FUNCTION_BLOCK FB_BMS
VAR_OUTPUT
	PowerStatus: eHVDC_Powerstatus := 0;
END_VAR
VAR_INPUT
	Set : st_BMS_Set;
END_VAR

VAR_OUTPUT
	BMSGet: st_BMS_GetStatus;
END_VAR

VAR	
	FBState				:	ePOUState;
	IO					:	FB_BMS_IO;
	HWControl			:	st_BMS_IO;
	
	InitTimeout			: 	TON := (PT:=T#3S);
	
	BMS_230V_StartupTimer : TON := (PT := TIME#3S0MS);
	BMS_24V_StartupTimer : TON := (PT := TIME#2S0MS);
	
	TempVar				: WORD;
	SFCInit				: BOOL := FALSE;
	SFCReset			: BOOL := FALSE;
	
//	by_CommErrorCounter	:	BYTE	:=	0;
	b_MBComErrorActive	: 	BOOL 	:= FALSE;
	
	ResetBMS	:	Bool; 
	b_BMSShutdownRequested: BOOL;
	
	BMSReadIntervalTimer	 : TON := (PT := TIME#1S0MS);
END_VAR

(*
FB_BMS

Inputs
	Set.b_EnableBMS				:	BOOL;
		Start BMS SFC sequence and initializes BMS. False means full BMS powerdown, so no status logging.
		With HVDC enabled, setting this value to False has no effect. Only after HVDC powerdown this value is tested.
		
	Set.b_ClearFault				:	BOOL;
		Clear errors and warning in BMS system. Set to true to initiate reset. Value resets automatically to false.
	
	Set.b_HVDC_Required			: 	BOOL;
		Set by FB_internalPowersupply. True initiates and keeps HVDC on, False initiates and retains powerdown

Outputs
	BMSGET
		-Some general status info
		-BATTinfo	struct with main operation battery data
		-MBMU_Status 	struct with detailed MBMU data
		-SBMU			Struct with detailed data per SBMU
		-Events			Warnings & Errors as per Sunspec list.
*)

IO(HWControl:=HWControl);

BMSReadIntervalTimer(in:= not BMSReadIntervalTimer.Q);

//Reset ErrorActive before entering SFC. 
//any remaining error in the Modbus methods will set Erroractive again. 
//This is pushed to events in BMS_Diagnostics

//TEMPBMSHB();
//hv required not allowed if BMS not enabled
set.b_HVDC_Required := set.b_HVDC_Required AND Set.b_EnableBMS;
//shutdown allowed if hvdc is offline
b_BMSShutdownRequested := (NOT Set.b_EnableBMS) AND BMSGet.BattInfo.ui_BMS_PowerOnStatus <> ePowerOnStatus.On; 

//b_MBComErrorActive := FALSE;

IF FBState = ePOUState.EMSTOP THEN
	Set.b_HVDC_Required := FALSE;
END_IF

BMSSFC();


IF ResetBMS THEN
	Reset();
END_IF


BMS_Diagnostics();

ACTION aBMSPoweroff:
HWControl.b_BMS_230V_Enable := FALSE;
HWControl.b_BMS_24V_Enable := FALSE;

BMSGet.BattInfo.b_BMSHeartBeatOK := FALSE;
BMSGet.BattInfo.ui_BMS_PowerOnStatus := ePowerOnStatus.Off;
BMSGet.BattInfo.ui_BMS_Status := eBMS_Status.Off;

BMSGet.MBMU_Status.BatteryStatus.b_BMSHeartBeatOK := FALSE;
BMSGet.MBMU_Status.BatteryStatus.ui_BMS_PowerOnStatus := ePowerOnStatus.Off;
BMSGet.MBMU_Status.BatteryStatus.ui_BMS_Status := eBMS_Status.Off;

FBState := ePOUState.OFF;
END_ACTION

ACTION aBMSPowerOn:

//230V inverter requires some startup time. Start this first to init SBMU before MBMU
//This may not be needed, but the idea is to make sure the MBMU can reach the SBMU's at boot.
FBState := ePOUState.PowerUp;
HWControl.b_BMS_230V_Enable := TRUE;
BMS_230V_StartupTimer(IN:=HWControl.b_BMS_230V_Enable);

HWControl.b_BMS_24V_Enable := BMS_230V_StartupTimer.Q;
BMS_24V_StartupTimer(IN:=HWControl.b_BMS_24V_Enable);
END_ACTION

ACTION aClearFaults:
SFCTip := ClearBMSFaults();
END_ACTION

ACTION aDisableInsulationMonitor:
SFCTip := OpenInsulationSwitch(TRUE);
END_ACTION

ACTION aGetMBMUData:
SFCTip := GetMBMUData();
END_ACTION

ACTION aGetSBMUData:
SFCTip := GetSBMUData();
END_ACTION

ACTION aGetStaticData:

IF (TempVar=0) THEN
	IF GetMBMUStaticSystemData() THEN
		TempVar:=1;
	END_IF;
ELSE
	IF GetSBMUStaticSystemData(TempVar) THEN
		TempVar := TempVar+1;
	END_IF
	
	IF TempVar > 4 then//BMSGet.MBMU_Status.by_NumberOfSubSystems THEN
		TempVar:=0;
		SFCTip := TRUE;
	END_IF
END_IF
END_ACTION

ACTION aGetStatus:
IF GetSystemStatus() THEN
	IF FBState = ePOUState.PowerUp THEN FBState := ePOUState.Init; END_IF
	SFCTip := TRUE;
END_IF
END_ACTION

ACTION aInit:
TempVar := 0;
SFCReset := false;
END_ACTION

ACTION aSetDateTime:
SFCTip := SetBMSDateTime();
END_ACTION

ACTION aSetPowerMode:
SFCTip := SetPowerMode();
END_ACTION

ACTION aWatchdog:
IF FBState = ePOUState.Init THEN FBState := ePOUState.Normal; END_IF

SFCTip := BMSHeartBeat();
TempVar := 0;
END_ACTION

METHOD BMS_Diagnostics : BOOL
VAR
	
END_VAR

BMSGet.Events.b_COMMUNICATION_ERROR				:=	BMSGet.MBMU_Status.GeneralSBMUStatus[6].5 	//SBMU CCAN comm lost
												OR BMSGet.MBMU_Status.GeneralSBMUStatus[6].6 	//SBMU SCAN comm lost
												OR BMSGet.MBMU_Status.GeneralSBMUStatus[6].7	//SBMU MCAN comm lost
												OR BMSGet.MBMU_Status.MBMUStatus[0].6			//MBMU MCAN comm warning
												OR BMSGet.MBMU_Status.MBMUStatus[0].7			//MBMU MCAN comm Lost
												OR BMSGet.MBMU_Status.MBMUStatus[0].8			//SBMU EMS COMM lost
												OR BMSGet.MBMU_Status.MBMUStatus[3].4			//SBMU MBMU comm fault
												OR b_MBComErrorActive;					//One or more Modbus communication errors 
									
BMSGet.Events.b_OVER_TEMP_ALARM					:= BMSGet.MBMU_Status.GeneralSBMUStatus[2].1;	//single cell Overtemperature warning 4

BMSGet.Events.b_OVER_TEMP_WARNING				:= BMSGet.MBMU_Status.GeneralSBMUStatus[1].14	//single cell Overtemperature warning 1
												OR BMSGet.MBMU_Status.GeneralSBMUStatus[2].0; 	//single cell Overtemperature warning 2

BMSGet.Events.b_UNDER_TEMP_ALARM				:= FALSE; //no data

BMSGet.Events.b_UNDER_TEMP_WARNING				:= BMSGet.MBMU_Status.GeneralSBMUStatus[2].2	//single cell Undertemperature warning 1
												OR BMSGet.MBMU_Status.GeneralSBMUStatus[2].3 	//single cell Undertemperature warning 2
												OR BMSGet.MBMU_Status.GeneralSBMUStatus[2].4; 	//single cell Undertemperature warning 3

BMSGet.Events.b_OVER_CHARGE_CURRENT_ALARM		:= BMSGet.MBMU_Status.GeneralSBMUStatus[1].9;	//Charge Overcurrent warning 4

BMSGet.Events.b_OVER_CHARGE_CURRENT_WARNING		:= BMSGet.MBMU_Status.GeneralSBMUStatus[1].6	//Charge Overcurrent warning 1
												OR BMSGet.MBMU_Status.GeneralSBMUStatus[1].7 	//Charge Overcurrent warning 2
												OR BMSGet.MBMU_Status.GeneralSBMUStatus[1].8; 	//Charge Overcurrent warning 3
											
BMSGet.Events.b_OVER_DISCHARGE_CURRENT_ALARM	:= BMSGet.MBMU_Status.GeneralSBMUStatus[1].5;	//Discharge Overcurrent warning 4

BMSGet.Events.b_OVER_DISCHARGE_CURRENT_WARNING	:= BMSGet.MBMU_Status.GeneralSBMUStatus[1].2	//Discharge Overcurrent warning 1
												OR BMSGet.MBMU_Status.GeneralSBMUStatus[1].3 	//Discharge Overcurrent warning 2
												OR BMSGet.MBMU_Status.GeneralSBMUStatus[1].4; 	//Discharge Overcurrent warning 3
											
BMSGet.Events.b_OVER_VOLT_ALARM					:= BMSGet.MBMU_Status.GeneralSBMUStatus[0].6;	//Single cell extreme overVoltage warning

BMSGet.Events.b_OVER_VOLT_WARNING				:= BMSGet.MBMU_Status.GeneralSBMUStatus[0].0	//Single cell overVoltage warning 1
												OR BMSGet.MBMU_Status.GeneralSBMUStatus[0].1 	//Single cell overVoltage warning 2
												OR BMSGet.MBMU_Status.GeneralSBMUStatus[0].2 	//Single cell overVoltage warning 3
												OR BMSGet.MBMU_Status.GeneralSBMUStatus[0].8 	//Single rack overVoltage warning 1
												OR BMSGet.MBMU_Status.GeneralSBMUStatus[0].9; 	//Single rack overVoltage warning 2
												
BMSGet.Events.b_UNDER_VOLT_ALARM				:= BMSGet.MBMU_Status.GeneralSBMUStatus[0].7;	//Single cell extreme underVoltage warning

BMSGet.Events.b_UNDER_VOLT_WARNING				:= BMSGet.MBMU_Status.GeneralSBMUStatus[0].3	//Single cell underVoltage warning 1
												OR BMSGet.MBMU_Status.GeneralSBMUStatus[0].4 	//Single cell underVoltage warning 2
												OR BMSGet.MBMU_Status.GeneralSBMUStatus[0].5 	//Single cell underVoltage warning 3
												OR BMSGet.MBMU_Status.GeneralSBMUStatus[0].10 	//Single rack underVoltage warning 1
												OR BMSGet.MBMU_Status.GeneralSBMUStatus[0].11; //Single rack underVoltage warning 2
												
BMSGet.Events.b_UNDER_SOC_MIN_ALARM				:= BMSGet.MBMU_Status.GeneralSBMUStatus[6].14;	//r_SOC low warning 2

BMSGet.Events.b_UNDER_SOC_MIN_WARNING			:= BMSGet.MBMU_Status.GeneralSBMUStatus[6].13;	//r_SOC low warning 1

BMSGet.Events.b_OVER_SOC_MAX_ALARM				:= FALSE; //no data

BMSGet.Events.b_OVER_SOC_MAX_WARNING			:= FALSE; //no data

BMSGet.Events.b_VOLTAGE_IMBALANCE_WARNING		:= BMSGet.MBMU_Status.GeneralSBMUStatus[0].12;	//large voltage difference warning

BMSGet.Events.b_TEMPERATURE_IMBALANCE_ALARM		:= FALSE; //no data
												
BMSGet.Events.b_TEMPERATURE_IMBALANCE_WARNING	:= BMSGet.MBMU_Status.GeneralSBMUStatus[2].5	//Large temperature difference warning 1
												OR BMSGet.MBMU_Status.GeneralSBMUStatus[2].6 	//Large temperature difference warning 2
												OR BMSGet.MBMU_Status.GeneralSBMUStatus[2].7; 	//Large temperature difference warning 3
												
BMSGet.Events.b_CONTACTOR_ERROR					:= BMSGet.MBMU_Status.GeneralSBMUStatus[5].1	//Main positive relay sticking
												OR BMSGet.MBMU_Status.GeneralSBMUStatus[5].2 	//Main negative relay sticking
												OR BMSGet.MBMU_Status.GeneralSBMUStatus[5].3 	//Both main relays sticking
												OR BMSGet.MBMU_Status.GeneralSBMUStatus[5].4 	//Main positive relay open
												OR BMSGet.MBMU_Status.GeneralSBMUStatus[5].5 	//Main negative relay open
												OR BMSGet.MBMU_Status.GeneralSBMUStatus[6].15; //HV open circuit warning
												
BMSGet.Events.b_FAN_ERROR						:= BMSGet.MBMU_Status.GeneralSBMUStatus[5].7;	//main control box fan warning

BMSGet.Events.b_GROUND_FAULT					:= FALSE; //no data

BMSGet.Events.b_OPEN_DOOR_ERROR					:= FALSE; //no data

BMSGet.Events.b_CURRENT_IMBALANCE_WARNING		:= FALSE; //no data

BMSGet.Events.b_OTHER_ALARM						:= BMSGet.MBMU_Status.GeneralSBMUStatus[0].13	//Invalid voltage warning
												OR BMSGet.MBMU_Status.GeneralSBMUStatus[1].10 	//Current sensor fault
												OR BMSGet.MBMU_Status.GeneralSBMUStatus[2].15 //single temperature sampling abnormal value warning
												OR BMSGet.MBMU_Status.GeneralSBMUStatus[3].0 	//multiple temperature sampling abnormal value warning
												OR BMSGet.MBMU_Status.GeneralSBMUStatus[4].9 	//CSC supply abnormal
												OR BMSGet.MBMU_Status.GeneralSBMUStatus[4].10 	//SBMU supply abnormal
												OR BMSGet.MBMU_Status.GeneralSBMUStatus[4].14 	//MSD warning
												OR BMSGet.MBMU_Status.GeneralSBMUStatus[4].15 	//rack fuse warning
												OR BMSGet.MBMU_Status.GeneralSBMUStatus[6].11 	//cell balance circuit short
												OR BMSGet.MBMU_Status.GeneralSBMUStatus[7].3 	//precharching failed twice
												OR BMSGet.MBMU_Status.MBMUStatus[1].7 			//estop fault
												OR BMSGet.MBMU_Status.MBMUStatus[3].3; 		//MBMU 24V fault
												
BMSGet.Events.b_OTHER_WARNING					:= BMSGet.MBMU_Status.MBMUStatus[0].0 			//insulation warning
												OR BMSGet.MBMU_Status.MBMUStatus[1].10 		//rack fan warning
												OR BMSGet.MBMU_Status.MBMUStatus[3].7;			//TMS warning
												
BMSGet.Events.b_CONFIGURATION_ALARM				:= BMSGet.MBMU_Status.GeneralSBMUStatus[5].0	//rack isolate switch warning
												OR BMSGet.MBMU_Status.GeneralSBMUStatus[5].6 	//battery rack door fault
												OR BMSGet.MBMU_Status.GeneralSBMUStatus[5].9 	//rack fire system level 1 fault
												OR BMSGet.MBMU_Status.GeneralSBMUStatus[5].10 	//smoke detector contact open
												OR BMSGet.MBMU_Status.GeneralSBMUStatus[5].11 	//temp detector contact open
												OR BMSGet.MBMU_Status.GeneralSBMUStatus[5].14 	//aerosol warning
												OR BMSGet.MBMU_Status.GeneralSBMUStatus[6].0 	//rack fire system level 2 fault
												OR BMSGet.MBMU_Status.GeneralSBMUStatus[6].10 	//SBMU TMS CCAN comm lost with hv on
												OR BMSGet.MBMU_Status.GeneralSBMUStatus[7].0 	//lvl 3 fault tms
												OR BMSGet.MBMU_Status.GeneralSBMUStatus[7].1 	//TMS mode conflict
												OR BMSGet.MBMU_Status.GeneralSBMUStatus[7].2 	//TMS warning
												OR BMSGet.MBMU_Status.GeneralSBMUStatus[8].0 	//Thermal runaway caused fire
												OR BMSGet.MBMU_Status.MBMUStatus[0].1	 		//Insulation fault
												OR BMSGet.MBMU_Status.MBMUStatus[0].2			//Insulation error
												OR BMSGet.MBMU_Status.MBMUStatus[0].3 			//Less HV racks than expected
												OR BMSGet.MBMU_Status.MBMUStatus[0].9			//IMM comm fault
												OR BMSGet.MBMU_Status.MBMUStatus[0].10 		//Air conditioning comm fault
												OR BMSGet.MBMU_Status.MBMUStatus[0].11			//TMS comm fault
												OR BMSGet.MBMU_Status.MBMUStatus[0].13			//TMS comm fault lvl 2
												OR BMSGet.MBMU_Status.MBMUStatus[0].14 		//TMS mode conflict
												OR BMSGet.MBMU_Status.MBMUStatus[0].15			//TMS comm fault level 1
												OR BMSGet.MBMU_Status.MBMUStatus[1].3	 		//AUX power DCDC failure
												OR BMSGet.MBMU_Status.MBMUStatus[1].4			//Fire system fault lvl 1
												OR BMSGet.MBMU_Status.MBMUStatus[1].5 			//Fire system fault lvl 2
												OR BMSGet.MBMU_Status.MBMUStatus[1].6			//Fire system failure warning
												OR BMSGet.MBMU_Status.MBMUStatus[1].8	 		//client estop fault
												OR BMSGet.MBMU_Status.MBMUStatus[1].9			//rack door fault
												OR BMSGet.MBMU_Status.MBMUStatus[1].12;		//smoke ex fan body fault
								
BMSGet.Events.b_CONFIGURATION_WARNING			:= BMSGet.MBMU_Status.GeneralSBMUStatus[6].8	//SBMU TMS CCAN comm lost
												OR BMSGet.MBMU_Status.MBMUStatus[0].12	 		//TMS comm warning
												OR BMSGet.MBMU_Status.MBMUStatus[1].0			//SPD failure
												OR BMSGet.MBMU_Status.MBMUStatus[1].1 			//Aux power DCDC failure
												OR BMSGet.MBMU_Status.MBMUStatus[1].2			//AUX power DCDC failure
												OR BMSGet.MBMU_Status.MBMUStatus[1].6 			//Fire system failure warning
												OR BMSGet.MBMU_Status.MBMUStatus[1].11;		//Smoke exhaust fan body warning
END_METHOD

METHOD BMSHeartBeat : BOOL

VAR_INST
	WriteReg		:	FB_MBWriteSingleReg;
	ReadReg			:	FB_MBReadRegs;
	
	readbCommBusy		:	BOOL;
	readbComError		:	BOOL;
	readerrID			:	UDINT;
	
	WritebCommBusy		:	BOOL;
	WritebComError		:	BOOL;
	WriteerrID			:	UDINT;
	
	ReadDone			:	F_Trig;
	ReadOK				: 	BOOL;
	WriteDone			:	F_Trig;
	WriteOK				: 	BOOL;
	
	ComTimer		:	Ton := (PT := TIME#0S200MS);
	
	OldValue		:	WORD := 0;
	BMSHBValue		:	WORD := 0;
	
	WatchdogUpdateTimer	:	Tof := (PT := TIME#3S0MS);
	WatchdogCommTimer	:	Tof := (PT := TIME#3S0MS);
	
	ComRetryCounter	:	USINT := 0;
END_VAR

ComTimer(in := NOT(ComTimer.Q));

ReadReg(
sIPAddr := Config.IP_BMS,
nTCPPort := Config.MBPort_BMS,
nUnitID := 255,//16#FF;
nMBAddr := 768,
nQuantity := 1,
cbLength := 2,
pDestAddr := ADR(BMSHBValue),
bExecute := ComTimer.Q,
tTimeout := T#100MS,
bBusy => readbCommBusy,
bError => readbComError,
nErrId => readerrID,
cbRead => 
);

ReadDone(clk := readbCommBusy);
ReadOK := ReadDone.Q AND NOT readbComError;


//read value is transmitted back into the write buffer if read is succesful
//BMS increments this value every second.
WriteReg(
sIPAddr := Config.IP_BMS,
nTCPPort := Config.MBPort_BMS,
nUnitID := 255,//16#FF;
nMBAddr := 896,
nValue := BMSHBValue,
tTimeout := T#100MS,
bExecute := ReadOK,
bBusy => WritebCommBusy,
bError => WritebComError,
nErrId => WriteerrID,
);

WriteDone(clk := writebCommBusy);
WriteOK := writeDone.Q AND NOT writebComError;

//if written value and BMS value are equal for longer than 3 seconds, the BMS isn't incrementing the value anymore or communication failed.
//BMS itself will throw warning after 30s and disable 10s after that.
WatchdogUpdateTimer(in:= (OldValue <> BMSHBValue));
OldValue := BMSHBValue;

//if modbus communication throws an error retry for 3s, otherwise system failed.
//WatchdogCommTimer(in:= WriteOK);

//both values are normally high and fall away if they timeout
BMSGet.BattInfo.b_BMSHeartBeatOK := WatchdogUpdateTimer.Q;// OR WatchdogCommTimer.Q;
BMSGet.MBMU_Status.BatteryStatus.b_BMSHeartBeatOK := WatchdogUpdateTimer.Q;

IF (ReadDone.Q AND readbComError) OR (WriteDone.Q AND WritebComError) THEN
	ComRetryCounter := ComRetryCounter + 1;
	IF COMRetryCounter > 5 THEN
		b_MBComErrorActive := TRUE;
		BMSGet.BattInfo.b_BMSHeartBeatOK := FALSE;
	END_IF
END_IF

IF WriteOK THEN
	ComRetryCounter := 0;
	BMSHeartBeat := TRUE;
END_IF
END_METHOD

ACTION BMSSFC:
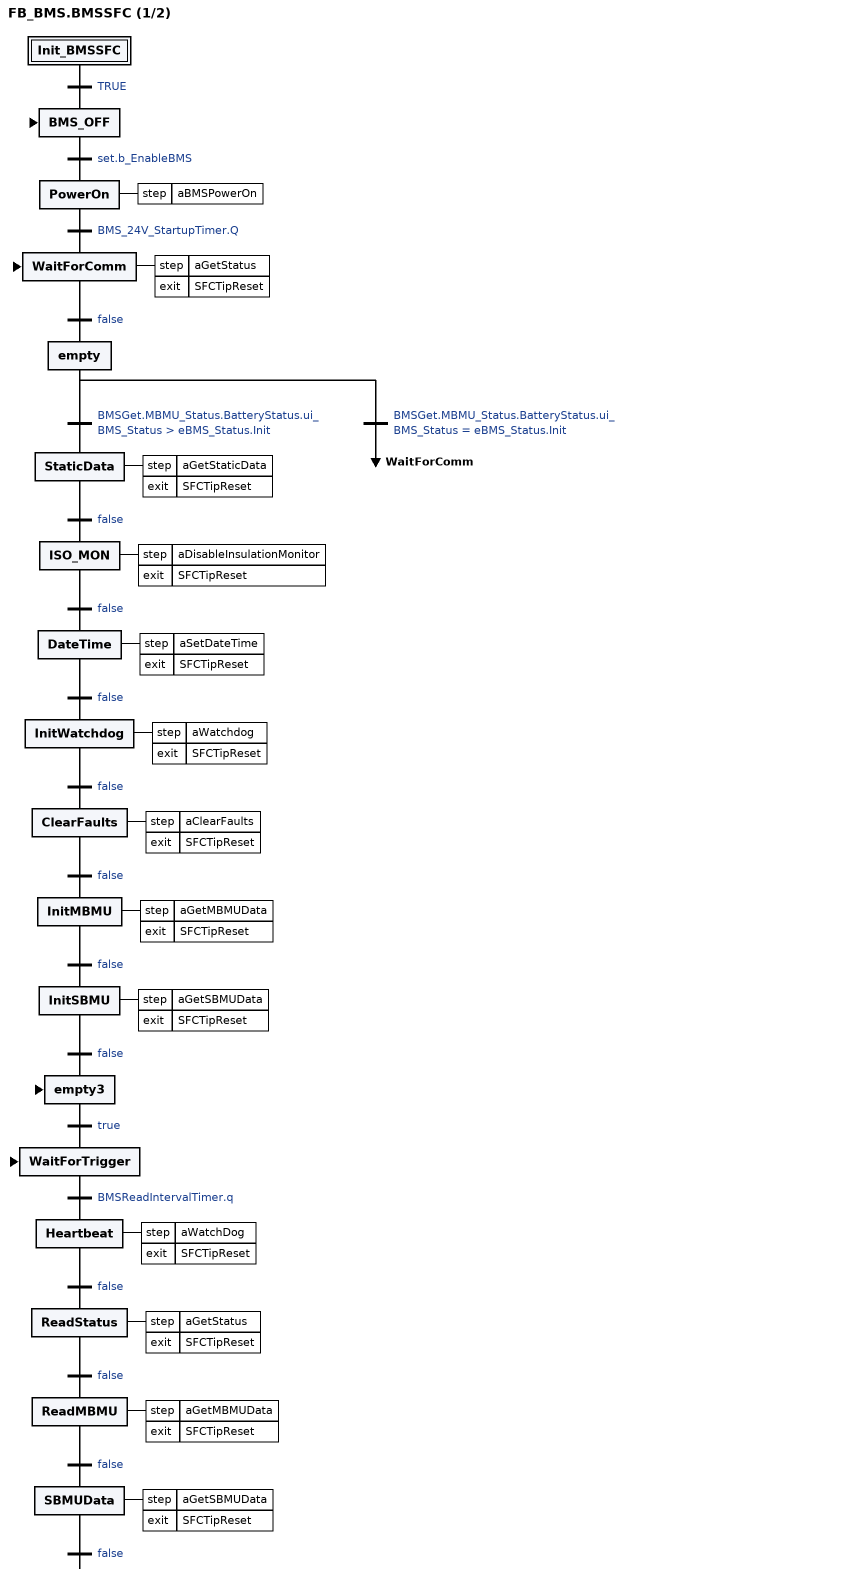
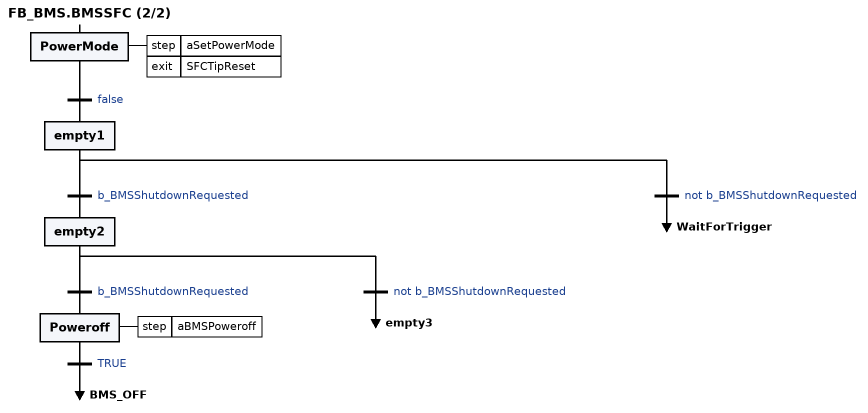
INITIAL_STEP Init_BMSSFC:
END_STEP
TRANSITION FROM Init_BMSSFC TO BMS_OFF
    := TRUE;
END_TRANSITION
STEP BMS_OFF:
END_STEP
TRANSITION FROM BMS_OFF TO PowerOn
    := set.b_EnableBMS;
END_TRANSITION
// macro BMSInit begins
STEP PowerOn:
    aBMSPowerOn(N);  // step action
END_STEP
TRANSITION FROM PowerOn TO WaitForComm
    := BMS_24V_StartupTimer.Q;
END_TRANSITION
STEP WaitForComm:
    aGetStatus(N);  // step action
    SFCTipReset(P0);  // exit action
END_STEP
TRANSITION FROM WaitForComm TO empty
    := false;
END_TRANSITION
STEP empty:
END_STEP
TRANSITION FROM empty TO StaticData
    := BMSGet.MBMU_Status.BatteryStatus.ui_BMS_Status > eBMS_Status.Init;
END_TRANSITION
TRANSITION FROM empty TO WaitForComm
    := BMSGet.MBMU_Status.BatteryStatus.ui_BMS_Status = eBMS_Status.Init;
END_TRANSITION
STEP StaticData:
    aGetStaticData(N);  // step action
    SFCTipReset(P0);  // exit action
END_STEP
TRANSITION FROM StaticData TO ISO_MON
    := false;
END_TRANSITION
STEP ISO_MON:
    aDisableInsulationMonitor(N);  // step action
    SFCTipReset(P0);  // exit action
END_STEP
TRANSITION FROM ISO_MON TO DateTime
    := false;
END_TRANSITION
STEP DateTime:
    aSetDateTime(N);  // step action
    SFCTipReset(P0);  // exit action
END_STEP
TRANSITION FROM DateTime TO InitWatchdog
    := false;
END_TRANSITION
STEP InitWatchdog:
    aWatchdog(N);  // step action
    SFCTipReset(P0);  // exit action
END_STEP
TRANSITION FROM InitWatchdog TO ClearFaults
    := false;
END_TRANSITION
STEP ClearFaults:
    aClearFaults(N);  // step action
    SFCTipReset(P0);  // exit action
END_STEP
TRANSITION FROM ClearFaults TO InitMBMU
    := false;
END_TRANSITION
STEP InitMBMU:
    aGetMBMUData(N);  // step action
    SFCTipReset(P0);  // exit action
END_STEP
TRANSITION FROM InitMBMU TO InitSBMU
    := false;
END_TRANSITION
STEP InitSBMU:
    aGetSBMUData(N);  // step action
    SFCTipReset(P0);  // exit action
END_STEP
TRANSITION FROM InitSBMU TO empty3
    := false;
END_TRANSITION
STEP empty3:
END_STEP
TRANSITION FROM empty3 TO WaitForTrigger
    := true;
END_TRANSITION
// macro BMSActive begins
STEP WaitForTrigger:
END_STEP
TRANSITION FROM WaitForTrigger TO Heartbeat
    := BMSReadIntervalTimer.q;
END_TRANSITION
STEP Heartbeat:
    aWatchDog(N);  // step action
    SFCTipReset(P0);  // exit action
END_STEP
TRANSITION FROM Heartbeat TO ReadStatus
    := false;
END_TRANSITION
STEP ReadStatus:
    aGetStatus(N);  // step action
    SFCTipReset(P0);  // exit action
END_STEP
TRANSITION FROM ReadStatus TO ReadMBMU
    := false;
END_TRANSITION
STEP ReadMBMU:
    aGetMBMUData(N);  // step action
    SFCTipReset(P0);  // exit action
END_STEP
TRANSITION FROM ReadMBMU TO SBMUData
    := false;
END_TRANSITION
STEP SBMUData:
    aGetSBMUData(N);  // step action
    SFCTipReset(P0);  // exit action
END_STEP
TRANSITION FROM SBMUData TO PowerMode
    := false;
END_TRANSITION
STEP PowerMode:
    aSetPowerMode(N);  // step action
    SFCTipReset(P0);  // exit action
END_STEP
TRANSITION FROM PowerMode TO empty1
    := false;
END_TRANSITION
STEP empty1:
END_STEP
TRANSITION FROM empty1 TO empty2
    := b_BMSShutdownRequested;
END_TRANSITION
TRANSITION FROM empty1 TO WaitForTrigger
    := not b_BMSShutdownRequested;
END_TRANSITION
STEP empty2:
END_STEP
TRANSITION FROM empty2 TO Poweroff
    := b_BMSShutdownRequested;
END_TRANSITION
TRANSITION FROM empty2 TO empty3
    := not b_BMSShutdownRequested;
END_TRANSITION
STEP Poweroff:
    aBMSPoweroff(N);  // step action
END_STEP
TRANSITION FROM Poweroff TO BMS_OFF
    := TRUE;
END_TRANSITION
// branch label Branch1_BMSSFC
// branch label Branch0_BMSSFC
END_ACTION

METHOD ClearBMSFaults : BOOL
VAR_INST
	WriteRegSet		:	FB_MBWriteSingleReg;
	WriteRegClear	:	FB_MBWriteSingleReg;
	ComTimer	:	Ton := (PT := TIME#200MS);
	
	bCommBusy	:	BOOL;
	bComError	:	BOOL;
	errID		:	UDINT;
	b_ClearDone	:	BOOL := FALSE;

	w_ClearFault	:	WORD;
	TX1Done 	: 	f_trig;
	
	bCommBusy2	:	BOOL;
	bComError2	:	BOOL;
	errID2		:	UDINT;
	TX2Done 	: 	f_trig;

	ComRetryCounter	:	USINT := 0;	
END_VAR
//Catl says we need to write 1 to clear, then write back to 0 to be able to log new errors.
//This method is called continuously when bms is active. It will usually write zero's.
//If set.b_ClearFault is 1, that will be written. The value will be cleared by this method after the write so next write will be a 0 again.
//With this, a reset cycle takes half a second with the current ComTimer.

ClearBMSFaults := FALSE;

ComTimer(in := NOT(ComTimer.Q));

//first write clearing register to 1
WriteRegSet(
	sIPAddr := Config.IP_BMS,
	nTCPPort := Config.MBPort_BMS,
	nUnitID := 255,//16#FF;
	nMBAddr := 908,
	nValue := 1,
	tTimeout := T#100MS,
	bExecute := ComTimer.Q,
	bBusy => bCommBusy,
	bError => bComError,
	nErrId => errID,
);

TX1Done(CLK := bCommBusy);
b_ClearDone	:= 	TX1Done.Q AND NOT bComError;

//reset value back to 0 afterwards. CATL requirement
WriteRegClear(
	sIPAddr := Config.IP_BMS,
	nTCPPort := Config.MBPort_BMS,
	nUnitID := 255,//16#FF;
	nMBAddr := 908,
	nValue := 0,
	tTimeout := T#100MS,
	bExecute := b_ClearDone,
	bBusy => bCommBusy2,
	bError => bComError2,
	nErrId => errID2
);

TX2Done(CLK := bCommBusy2);

IF (TX1Done.Q AND bComError) OR (TX2Done.Q AND bComError2) THEN
	ComRetryCounter := ComRetryCounter + 1;
	IF COMRetryCounter > 5 THEN
		b_MBComErrorActive := TRUE;
	END_IF
END_IF

IF TX2Done.Q AND NOT bComError2 THEN
	ComRetryCounter := 0;
	ClearBMSFaults := TRUE;
END_IF
END_METHOD

METHOD EMSTOP : BOOL
VAR_INPUT
	EMSTOP_Active	:	BOOL;
END_VAR
EMSTOP := FALSE;

FBState := ePOUState.EMSTOP;
set.b_HVDC_Required := FALSE;

IF BMSGet.BattInfo.ui_BMS_PowerOnStatus = ePowerOnStatus.Off THEN
	EMSTOP := TRUE;
END_IF
END_METHOD

METHOD GetCellData : BOOL
VAR_INPUT
	SBMUID	:	BYTE;	//SBMU 1-#ofstrings
	CSCID	:	BYTE;	//CSC 1-4
END_VAR

VAR_OUTPUT
	CellVoltages		:	ARRAY[1..52] OF REAL;
	Celltemperatures	:	ARRAY[1..16] OF INT;
	BalanceStatus		:	ARRAY[1..4] OF WORD; //bit per cell?
END_VAR

VAR_INST
	MBReadCellVoltages	: 	FB_MBReadRegs;
	MBReadTemperatures	: 	FB_MBReadRegs;
	MBReadCellBalance	: 	FB_MBReadRegs;
	
//	CellVoltageData		: 	ARRAY[1..52] OF WORD;
	TemperatureData		: 	ARRAY[1..16] OF BYTE;
//	CellBalanceData		: 	ARRAY[1..4] OF WORD;
	
	bCommBusy			:	ARRAY[1..3] OF BOOL;
	bComError			:	ARRAY[1..3] OF BOOL;
	errID				:	ARRAY[1..3] OF UDINT;
	cbRead				:	ARRAY[1..3] OF UDINT;
	TransmissionDone	: 	ARRAY[1..3] OF f_trig;
	
	DataComplete		:	ARRAY[1..3] OF BOOL;
	
	ComTimer			:	Ton := (PT := TIME#0S500MS);
END_VAR

VAR
	LoopCounter			:	INT;
END_VAR

GetCellData := FALSE;

IF (SBMUID < 1) OR (SBMUID > BMSGet.MBMU_Status.by_NumberOfSubSystems) THEN
	GetCellData := TRUE;
	RETURN;
END_IF
IF (CSCID < 1) OR (CSCID > 4) THEN
	GetCellData := TRUE;
	RETURN;
END_IF

ComTimer(in := NOT(ComTimer.Q));

IF ComTimer.Q THEN
	DataComplete[1] := FALSE;
	DataComplete[2] := FALSE;
	DataComplete[3] := FALSE;
END_IF

MBReadCellVoltages(
sIPAddr := Config.IP_BMS,
nTCPPort := Config.MBPort_BMS,
nUnitID := 255,//16#FF;
nMBAddr := (SBMUID*1024)+128+(52*(CSCID-1)),	//SBMU 1, module 1, start at 0x0480, increment 52 per module & 1024 per sbmu
nQuantity := 52,
cbLength := SIZEOF(CellVoltages),
pDestAddr := ADR(CellVoltages),
bExecute := ComTimer.Q,
bBusy => bCommBusy[1],
bError => bComError[1],
nErrId => errID[1],
cbRead => cbRead[1]
);

MBReadTemperatures(
sIPAddr := Config.IP_BMS,
nTCPPort := Config.MBPort_BMS,
nUnitID := 1,//16#FF;
nMBAddr := (SBMUID*1024)+704+(8*(CSCID-1)),	//SBMU 1, module 1, start at 0x06c0, increment 8 (16 byte) per module & 1024 per sbmu
nQuantity := 8*2,
cbLength := SIZEOF(TemperatureData),
pDestAddr := ADR(TemperatureData),
bExecute := ComTimer.Q,
bBusy => bCommBusy[2],
bError => bComError[2],
nErrId => errID[2],
cbRead => cbRead[2]
);

MBReadTemperatures(
sIPAddr := Config.IP_BMS,
nTCPPort := Config.MBPort_BMS,
nUnitID := 1,//16#FF;
nMBAddr := (SBMUID*1024)+912+(4*(CSCID-1)),	//SBMU 1, module 1, start at 0x0790, increment 4 per module & 1024 per sbmu
											//not sure if CSC2 starts at address 4, or immediatly follows after last cell of csc1.
nQuantity := 4*2,
cbLength := SIZEOF(BalanceStatus),
pDestAddr := ADR(BalanceStatus),
bExecute := ComTimer.Q,
bBusy => bCommBusy[3],
bError => bComError[3],
nErrId => errID[3],
cbRead => cbRead[3]
);

TransmissionDone[1](clk:=bCommBusy[1]);
TransmissionDone[2](clk:=bCommBusy[2]);
TransmissionDone[3](clk:=bCommBusy[3]);

IF TransmissionDone[1].Q AND NOT bComError[1] THEN
	DataComplete[1] := TRUE;
END_IF

IF TransmissionDone[2].Q AND NOT bComError[2] THEN
	FOR loopcounter := 1 TO 16 BY 1 DO
		Celltemperatures[loopcounter] := TemperatureData[loopcounter]-50;
	END_FOR
	DataComplete[2] := TRUE;
END_IF

IF TransmissionDone[1].Q AND NOT bComError[1] THEN
	DataComplete[3] := TRUE;
END_IF

GetCellData := DataComplete[1] AND DataComplete[2] AND DataComplete[3];
END_METHOD

METHOD GetDiagnostics 
VAR_IN_OUT
	AddError		: ARRAY [*] OF FB_AddErrorST;
	a_ActiveEvents	: ARRAY [*] OF ST_ErrorStruct;
	w_Index			: WORD;
END_VAR

VAR_OUTPUT
	b_errorActive	: BOOL;
	b_warningActive	: BOOL;
END_VAR

VAR
	by_errCt	: BYTE;
	by_warnCt	: BYTE;
	w_ID		: WORD;
END_VAR
(*BMS errors (sunspec)*)
	(*BMS Communication error*)		AddError[w_Index](
			in_b_ErrorTrig			:= BMSGet.Events.b_COMMUNICATION_ERROR,
			out_ST_Error			:= a_ActiveEvents[w_Index],
			w_ID					:= 1 + w_ID,
			s_Message				:= 'BMS communication error',
			e_sev					:= eSeverity.EmergencyShutdown,	//<-- maybe normal shutdown?
			in_b_AutoClear			:= FALSE,
			in_t_TriggerTime		:= TIME#1000MS,
			//in_e_ErrAckAccess		:= TRUE,
			);
		IF AddError[w_Index].b_out THEN by_errCt := by_errCt + 1; END_IF;
		w_Index := w_Index +1;
		
	(*Configuration fault*)		AddError[w_Index](
			in_b_ErrorTrig			:= BMSGet.Events.b_CONFIGURATION_ALARM,
			out_ST_Error			:= a_ActiveEvents[w_Index],
			w_ID					:= 1 + w_ID,
			s_Message				:= 'BMS configuration error',
			e_sev					:= eSeverity.NormalShutdown,
			in_b_AutoClear			:= FALSE,
			//in_t_TriggerTime		:= TIME#500MS,
			//in_e_ErrAckAccess		:= TRUE,
			);
		IF AddError[w_Index].b_out THEN by_errCt := by_errCt + 1; END_IF;
		w_Index := w_Index +1;
	
	(*Configuration warning*)		AddError[w_Index](
			in_b_ErrorTrig			:= BMSGet.Events.b_CONFIGURATION_WARNING,
			out_ST_Error			:= a_ActiveEvents[w_Index],
			w_ID					:= 1 + w_ID,
			s_Message				:= 'BMS configuration error',
			e_sev					:= eSeverity.Warning,
			in_b_AutoClear			:= FALSE,
			//in_t_TriggerTime		:= TIME#500MS,
			//in_e_ErrAckAccess		:= TRUE,
			);
		IF AddError[w_Index].b_out THEN by_errCt := by_errCt + 1; END_IF;
		w_Index := w_Index +1;
		
	(*Contactor fault*)		AddError[w_Index](
			in_b_ErrorTrig			:= BMSGet.Events.b_CONTACTOR_ERROR,
			out_ST_Error			:= a_ActiveEvents[w_Index],
			w_ID					:= 1 + w_ID,
			s_Message				:= 'BMS Contactor fault',
			e_sev					:= eSeverity.EmergencyShutdown,
			in_b_AutoClear			:= FALSE,
			//in_t_TriggerTime		:= TIME#500MS,
			//in_e_ErrAckAccess		:= TRUE,
			);
		IF AddError[w_Index].b_out THEN by_errCt := by_errCt + 1; END_IF;
		w_Index := w_Index +1;
		
	(*Current imbalance warning*)		AddError[w_Index](						//unused, will always be false
			in_b_ErrorTrig			:= BMSGet.Events.b_CURRENT_IMBALANCE_WARNING,
			out_ST_Error			:= a_ActiveEvents[w_Index],
			w_ID					:= 1 + w_ID,
			s_Message				:= 'BMS Current imbalance warning',
			e_sev					:= eSeverity.Warning,
			in_b_AutoClear			:= FALSE,
			//in_t_TriggerTime		:= TIME#500MS,
			//in_e_ErrAckAccess		:= TRUE,
			);
		IF AddError[w_Index].b_out THEN by_errCt := by_errCt + 1; END_IF;
		w_Index := w_Index +1;
		
	(*Fan error*)		AddError[w_Index](
			in_b_ErrorTrig			:= BMSGet.Events.b_FAN_ERROR,
			out_ST_Error			:= a_ActiveEvents[w_Index],
			w_ID					:= 1 + w_ID,
			s_Message				:= 'BMS fan error',
			e_sev					:= eSeverity.NormalShutdown,
			in_b_AutoClear			:= FALSE,
			//in_t_TriggerTime		:= TIME#500MS,
			//in_e_ErrAckAccess		:= TRUE,
			);
		IF AddError[w_Index].b_out THEN by_errCt := by_errCt + 1; END_IF;
		w_Index := w_Index +1;

	(*Ground fault*)		AddError[w_Index](
			in_b_ErrorTrig			:= BMSGet.Events.b_GROUND_FAULT,		//unused, will always be false
			out_ST_Error			:= a_ActiveEvents[w_Index],
			w_ID					:= 1 + w_ID,
			s_Message				:= 'BMS Insulation fault',
			e_sev					:= eSeverity.EmergencyShutdown,
			in_b_AutoClear			:= FALSE,
			//in_t_TriggerTime		:= TIME#500MS,
			//in_e_ErrAckAccess		:= TRUE,
			);
		IF AddError[w_Index].b_out THEN by_errCt := by_errCt + 1; END_IF;
		w_Index := w_Index +1;

	(*Door open error*)		AddError[w_Index](							//unused, will always be false
			in_b_ErrorTrig			:= BMSGet.Events.b_OPEN_DOOR_ERROR,
			out_ST_Error			:= a_ActiveEvents[w_Index],
			w_ID					:= 1 + w_ID,
			s_Message				:= 'BMS door open',
			e_sev					:= eSeverity.NormalShutdown,
			in_b_AutoClear			:= FALSE,
			//in_t_TriggerTime		:= TIME#500MS,
			//in_e_ErrAckAccess		:= TRUE,
			);
		IF AddError[w_Index].b_out THEN by_errCt := by_errCt + 1; END_IF;
		w_Index := w_Index +1;

	(*misc alarm*)		AddError[w_Index](							
			in_b_ErrorTrig			:= BMSGet.Events.b_OTHER_ALARM,
			out_ST_Error			:= a_ActiveEvents[w_Index],
			w_ID					:= 1 + w_ID,
			s_Message				:= 'BMS miscellaneous error',
			e_sev					:= eSeverity.NormalShutdown,
			in_b_AutoClear			:= FALSE,
			//in_t_TriggerTime		:= TIME#500MS,
			//in_e_ErrAckAccess		:= TRUE,
			);
		IF AddError[w_Index].b_out THEN by_errCt := by_errCt + 1; END_IF;
		w_Index := w_Index +1;
		
	(*misc warning*)		AddError[w_Index](							
			in_b_ErrorTrig			:= BMSGet.Events.b_OTHER_WARNING,
			out_ST_Error			:= a_ActiveEvents[w_Index],
			w_ID					:= 1 + w_ID,
			s_Message				:= 'BMS miscellaneous warning',
			e_sev					:= eSeverity.Warning,
			in_b_AutoClear			:= FALSE,
			//in_t_TriggerTime		:= TIME#500MS,
			//in_e_ErrAckAccess		:= TRUE,
			);
		IF AddError[w_Index].b_out THEN by_errCt := by_errCt + 1; END_IF;
		w_Index := w_Index +1;

	(*Overcharge current alarm*)		AddError[w_Index](							
			in_b_ErrorTrig			:= BMSGet.Events.b_OVER_CHARGE_CURRENT_ALARM,
			out_ST_Error			:= a_ActiveEvents[w_Index],
			w_ID					:= 1 + w_ID,
			s_Message				:= 'BMS Charge current too high error',
			e_sev					:= eSeverity.NormalShutdown,			
			in_b_AutoClear			:= FALSE,									
			//in_t_TriggerTime		:= TIME#500MS,
			//in_e_ErrAckAccess		:= TRUE,
			);
		IF AddError[w_Index].b_out THEN by_errCt := by_errCt + 1; END_IF;
		w_Index := w_Index +1;
		
	(*Overcharge current warning*)		AddError[w_Index](							
			in_b_ErrorTrig			:= BMSGet.Events.b_OVER_CHARGE_CURRENT_WARNING,
			out_ST_Error			:= a_ActiveEvents[w_Index],
			w_ID					:= 1 + w_ID,
			s_Message				:= 'BMS Charge current too high warning',
			e_sev					:= eSeverity.Warning,				//<-- Powerstack should lower the power
			in_b_AutoClear			:= FALSE,								
			//in_t_TriggerTime		:= TIME#500MS,
			//in_e_ErrAckAccess		:= TRUE,
			);
		IF AddError[w_Index].b_out THEN by_errCt := by_errCt + 1; END_IF;
		w_Index := w_Index +1;
		
	(*OverDischarge current Alarm*)		AddError[w_Index](							
			in_b_ErrorTrig			:= BMSGet.Events.b_OVER_DISCHARGE_CURRENT_ALARM,
			out_ST_Error			:= a_ActiveEvents[w_Index],
			w_ID					:= 1 + w_ID,
			s_Message				:= 'BMS Discharge current too high error',
			e_sev					:= eSeverity.NormalShutdown,				
			in_b_AutoClear			:= FALSE,								
			//in_t_TriggerTime		:= TIME#500MS,
			//in_e_ErrAckAccess		:= TRUE,
			);
			
		IF AddError[w_Index].b_out THEN by_errCt := by_errCt + 1; END_IF;
		w_Index := w_Index +1;
		
	(*OverDischarge current warning*)		AddError[w_Index](							
			in_b_ErrorTrig			:= BMSGet.Events.b_OVER_DISCHARGE_CURRENT_WARNING,
			out_ST_Error			:= a_ActiveEvents[w_Index],
			w_ID					:= 1 + w_ID,
			s_Message				:= 'BMS Discharge current too high warning',
			e_sev					:= eSeverity.Warning,				//<-- Powerstack should lower the power
			in_b_AutoClear			:= FALSE,								
			//in_t_TriggerTime		:= TIME#500MS,
			//in_e_ErrAckAccess		:= TRUE,
			);
		IF AddError[w_Index].b_out THEN by_errCt := by_errCt + 1; END_IF;
		w_Index := w_Index +1;
		
	(*Overcharge r_SOC error*)		AddError[w_Index](							//unused, will remain false
			in_b_ErrorTrig			:= BMSGet.Events.b_OVER_SOC_MAX_ALARM,
			out_ST_Error			:= a_ActiveEvents[w_Index],
			w_ID					:= 1 + w_ID,
			s_Message				:= 'BMS r_SOC too high error',
			e_sev					:= eSeverity.NormalShutdown,				
			in_b_AutoClear			:= FALSE,								
			//in_t_TriggerTime		:= TIME#500MS,
			//in_e_ErrAckAccess		:= TRUE,
			);
		IF AddError[w_Index].b_out THEN by_errCt := by_errCt + 1; END_IF;
		w_Index := w_Index +1;
		
	(*Overcharge r_SOC error*)		AddError[w_Index](							//unused, will remain false
			in_b_ErrorTrig			:= BMSGet.Events.b_OVER_SOC_MAX_WARNING,
			out_ST_Error			:= a_ActiveEvents[w_Index],
			w_ID					:= 1 + w_ID,
			s_Message				:= 'BMS r_SOC too high warning',
			e_sev					:= eSeverity.Warning,				
			in_b_AutoClear			:= FALSE,								
			//in_t_TriggerTime		:= TIME#500MS,
			//in_e_ErrAckAccess		:= TRUE,
			);
		IF AddError[w_Index].b_out THEN by_errCt := by_errCt + 1; END_IF;
		w_Index := w_Index +1;
		
	(*OverDischarge r_SOC error*)		AddError[w_Index](							
			in_b_ErrorTrig			:= BMSGet.Events.b_UNDER_SOC_MIN_ALARM,
			out_ST_Error			:= a_ActiveEvents[w_Index],
			w_ID					:= 1 + w_ID,
			s_Message				:= 'BMS r_SOC too low error',
			e_sev					:= eSeverity.NormalShutdown,				
			in_b_AutoClear			:= FALSE,								
			//in_t_TriggerTime		:= TIME#500MS,
			//in_e_ErrAckAccess		:= TRUE,
			);
		IF AddError[w_Index].b_out THEN by_errCt := by_errCt + 1; END_IF;
		w_Index := w_Index +1;
		
	(*OverDischarge r_SOC error*)		AddError[w_Index](							
			in_b_ErrorTrig			:= BMSGet.Events.b_UNDER_SOC_MIN_WARNING,
			out_ST_Error			:= a_ActiveEvents[w_Index],
			w_ID					:= 1 + w_ID,
			s_Message				:= 'BMS r_SOC too low warning',
			e_sev					:= eSeverity.Warning,				
			in_b_AutoClear			:= FALSE,								
			//in_t_TriggerTime		:= TIME#500MS,
			//in_e_ErrAckAccess		:= TRUE,
			);
		IF AddError[w_Index].b_out THEN by_errCt := by_errCt + 1; END_IF;
		w_Index := w_Index +1;
		
	(*OverTemperature error*)		AddError[w_Index](							
			in_b_ErrorTrig			:= BMSGet.Events.b_OVER_TEMP_ALARM,
			out_ST_Error			:= a_ActiveEvents[w_Index],
			w_ID					:= 1 + w_ID,
			s_Message				:= 'Battery Overtemperature error',
			e_sev					:= eSeverity.NormalShutdown,				
			in_b_AutoClear			:= FALSE,								
			//in_t_TriggerTime		:= TIME#500MS,
			//in_e_ErrAckAccess		:= TRUE,
			);
		IF AddError[w_Index].b_out THEN by_errCt := by_errCt + 1; END_IF;
		w_Index := w_Index +1;		

	(*OverTemperature warning*)		AddError[w_Index](							
			in_b_ErrorTrig			:= BMSGet.Events.b_OVER_TEMP_WARNING,
			out_ST_Error			:= a_ActiveEvents[w_Index],
			w_ID					:= 1 + w_ID,
			s_Message				:= 'Battery Overtemperature warning',
			e_sev					:= eSeverity.Warning,				
			in_b_AutoClear			:= FALSE,								
			//in_t_TriggerTime		:= TIME#500MS,
			//in_e_ErrAckAccess		:= TRUE,
			);
		IF AddError[w_Index].b_out THEN by_errCt := by_errCt + 1; END_IF;
		w_Index := w_Index +1;
	
	(*OverVoltage error*)		AddError[w_Index](							
			in_b_ErrorTrig			:= BMSGet.Events.b_OVER_VOLT_ALARM,
			out_ST_Error			:= a_ActiveEvents[w_Index],
			w_ID					:= 1 + w_ID,
			s_Message				:= 'Battery overvoltage error',
			e_sev					:= eSeverity.NormalShutdown,				
			in_b_AutoClear			:= FALSE,								
			//in_t_TriggerTime		:= TIME#500MS,
			//in_e_ErrAckAccess		:= TRUE,
			);
		IF AddError[w_Index].b_out THEN by_errCt := by_errCt + 1; END_IF;
		w_Index := w_Index +1;		

	(*OverVoltage warning*)		AddError[w_Index](							
			in_b_ErrorTrig			:= BMSGet.Events.b_OVER_VOLT_WARNING,
			out_ST_Error			:= a_ActiveEvents[w_Index],
			w_ID					:= 1 + w_ID,
			s_Message				:= 'Battery overvoltage warning',
			e_sev					:= eSeverity.Warning,				
			in_b_AutoClear			:= FALSE,								
			//in_t_TriggerTime		:= TIME#500MS,
			//in_e_ErrAckAccess		:= TRUE,
			);
		IF AddError[w_Index].b_out THEN by_errCt := by_errCt + 1; END_IF;
		w_Index := w_Index +1;
		
	(*Temperature imbalance error*)		AddError[w_Index](							
			in_b_ErrorTrig			:= BMSGet.Events.b_TEMPERATURE_IMBALANCE_ALARM,
			out_ST_Error			:= a_ActiveEvents[w_Index],
			w_ID					:= 1 + w_ID,
			s_Message				:= 'Battery temperature imbalance error',
			e_sev					:= eSeverity.NormalShutdown,				
			in_b_AutoClear			:= FALSE,								
			//in_t_TriggerTime		:= TIME#500MS,
			//in_e_ErrAckAccess		:= TRUE,
			);
		IF AddError[w_Index].b_out THEN by_errCt := by_errCt + 1; END_IF;
		w_Index := w_Index +1;		

	(*Temperature imbalance warning*)		AddError[w_Index](							
			in_b_ErrorTrig			:= BMSGet.Events.b_TEMPERATURE_IMBALANCE_WARNING,
			out_ST_Error			:= a_ActiveEvents[w_Index],
			w_ID					:= 1 + w_ID,
			s_Message				:= 'Battery temperature imbalance warning',
			e_sev					:= eSeverity.Warning,				
			in_b_AutoClear			:= FALSE,								
			//in_t_TriggerTime		:= TIME#500MS,
			//in_e_ErrAckAccess		:= TRUE,
			);
		IF AddError[w_Index].b_out THEN by_errCt := by_errCt + 1; END_IF;
		w_Index := w_Index +1;

	(*Under Temperature error*)		AddError[w_Index](							
			in_b_ErrorTrig			:= BMSGet.Events.b_UNDER_TEMP_ALARM,
			out_ST_Error			:= a_ActiveEvents[w_Index],
			w_ID					:= 1 + w_ID,
			s_Message				:= 'Battery temperature low error',
			e_sev					:= eSeverity.NormalShutdown,				
			in_b_AutoClear			:= FALSE,								
			//in_t_TriggerTime		:= TIME#500MS,
			//in_e_ErrAckAccess		:= TRUE,
			);
		IF AddError[w_Index].b_out THEN by_errCt := by_errCt + 1; END_IF;
		w_Index := w_Index +1;		

	(*Under Temperature warning*)		AddError[w_Index](							
			in_b_ErrorTrig			:= BMSGet.Events.b_UNDER_TEMP_WARNING,
			out_ST_Error			:= a_ActiveEvents[w_Index],
			w_ID					:= 1 + w_ID,
			s_Message				:= 'Battery temperature low warning',
			e_sev					:= eSeverity.Warning,				
			in_b_AutoClear			:= FALSE,								
			//in_t_TriggerTime		:= TIME#500MS,
			//in_e_ErrAckAccess		:= TRUE,
			);
		IF AddError[w_Index].b_out THEN by_errCt := by_errCt + 1; END_IF;
		w_Index := w_Index +1;

	(*Under Temperature error*)		AddError[w_Index](							
			in_b_ErrorTrig			:= BMSGet.Events.b_UNDER_VOLT_ALARM,
			out_ST_Error			:= a_ActiveEvents[w_Index],
			w_ID					:= 1 + w_ID,
			s_Message				:= 'Battery undervoltage error',
			e_sev					:= eSeverity.NormalShutdown,				
			in_b_AutoClear			:= FALSE,								
			//in_t_TriggerTime		:= TIME#500MS,
			//in_e_ErrAckAccess		:= TRUE,
			);
		IF AddError[w_Index].b_out THEN by_errCt := by_errCt + 1; END_IF;
		w_Index := w_Index +1;		

	(*Under Temperature warning*)		AddError[w_Index](							
			in_b_ErrorTrig			:= BMSGet.Events.b_UNDER_VOLT_WARNING,
			out_ST_Error			:= a_ActiveEvents[w_Index],
			w_ID					:= 1 + w_ID,
			s_Message				:= 'Battery undervoltage warning',
			e_sev					:= eSeverity.Warning,				
			in_b_AutoClear			:= FALSE,								
			//in_t_TriggerTime		:= TIME#500MS,
			//in_e_ErrAckAccess		:= TRUE,
			);
		IF AddError[w_Index].b_out THEN by_errCt := by_errCt + 1; END_IF;
		w_Index := w_Index +1;
		
	(*Battery voltage imbalance warning*)		AddError[w_Index](							
			in_b_ErrorTrig			:= BMSGet.Events.b_VOLTAGE_IMBALANCE_WARNING,
			out_ST_Error			:= a_ActiveEvents[w_Index],
			w_ID					:= 1 + w_ID,
			s_Message				:= 'Battery voltage imbalance warning',
			e_sev					:= eSeverity.Warning,				
			in_b_AutoClear			:= FALSE,								
			//in_t_TriggerTime		:= TIME#500MS,
			//in_e_ErrAckAccess		:= TRUE,
			);
		IF AddError[w_Index].b_out THEN by_errCt := by_errCt + 1; END_IF;
		w_Index := w_Index +1;
END_METHOD

METHOD GetMBMUData : BOOL
VAR_INST
	
	MBReadMBMU			: 	FB_MBReadRegs;
	MBMUData 			: 	ARRAY[0..52] OF WORD;
	bCommBusy			:	BOOL;
	bComError			:	BOOL;
	errID				:	UDINT;
	cbRead				:	UDINT;
	TransmissionDone	: 	f_trig;
	COMretryCounter		:	USINT := 0;
	
	ComTimer			:	Ton := (PT := TIME#0S200MS);
END_VAR

VAR
	Counter				:	INT;
END_VAR
//read mbmu data every 100ms

GetMBMUData := FALSE;

ComTimer(in := NOT(ComTimer.Q));

MBReadMBMU(
sIPAddr := Config.IP_BMS,
nTCPPort := Config.MBPort_BMS,
nUnitID := 255,//16#FF;
nMBAddr := 0,
nQuantity := 53,
cbLength := SIZEOF(MBMUData),
pDestAddr := ADR(MBMUData),
bExecute := ComTimer.Q,
bBusy => bCommBusy,
bError => bComError,
nErrId => errID,
cbRead => cbRead,
tTimeout := T#100MS
);

TransmissionDone(CLK := bCommBusy);

IF TransmissionDone.Q THEN
	IF NOT bComError THEN
		MEMCPY(ADR(BMSGet.MBMU_Status.GeneralSBMUStatus[0]), ADR(MBMUData[0]), 32);	//0x0000 - 0x000f
		MEMCPY(ADR(BMSGet.MBMU_Status.MBMUStatus[0]), ADR(MBMUData[16]), 32);			//0x0010 - 0x001f
	
		BMSGet.MBMU_Status.BatteryStatus.r_SystemVoltage := WORD_TO_REAL(MBMUData[32])/10; 						//0-1500V with 0.1V/bit
		BMSGet.MBMU_Status.BatteryStatus.r_SystemCurrent := WORD_TO_REAL(MBMUData[33])-20000; 					//-20k .. +20k kW in 1kW/bit steps
		
		BMSGet.MBMU_Status.BatteryStatus.r_SOC := WORD_TO_REAL(MBMUData[34])/10; 								//0-100% with 0.1%/bit;
		BMSGet.MBMU_Status.BatteryStatus.r_SOH := WORD_TO_REAL(MBMUData[35])/10; 								//0-100% with 0.1%/bit;
		
		BMSGet.MBMU_Status.BatteryStatus.CellVoltage[eSubValues.Maximum] := WORD_TO_REAL(MBMUData[36])/1000;	//0-5v with 0.001v/bit;
		BMSGet.MBMU_Status.BatteryStatus.CellVoltage[eSubValues.Minimum] := WORD_TO_REAL(MBMUData[37])/1000;	//0-5v with 0.001v/bit;
		BMSGet.MBMU_Status.BatteryStatus.CellVoltage[eSubValues.Average] := WORD_TO_REAL(MBMUData[38])/1000;	//0-5v with 0.001v/bit;
		
		BMSGet.MBMU_Status.BatteryStatus.CellTemperature[eSubValues.Maximum] := WORD_TO_REAL(MBMUData[39])-50;	//-50..200gr with 1gr/bit;
		BMSGet.MBMU_Status.BatteryStatus.CellTemperature[eSubValues.Minimum] := WORD_TO_REAL(MBMUData[40])-50;	//-50..200gr with 1gr/bit;
		BMSGet.MBMU_Status.BatteryStatus.CellTemperature[eSubValues.Average] := WORD_TO_REAL(MBMUData[41])-50;	//-50..200gr with 1gr/bit;
		
		BMSGet.MBMU_Status.BatteryStatus.r_MaxChargeCurrentAllowed := WORD_TO_REAL(MBMUData[42])-20000;			//-20k .. +20k A in 1A/bit steps
		BMSGet.MBMU_Status.BatteryStatus.r_MaxDischargeCurrentAllowed := WORD_TO_REAL(MBMUData[43])-20000;			//-20k .. +20k A in 1A/bit steps
		
		BMSGet.MBMU_Status.BatteryStatus.r_MaxChargePowerAllowed := WORD_TO_REAL(MBMUData[44])-20000;				//-20k .. +20k kW in 1kW/bit steps
		BMSGet.MBMU_Status.BatteryStatus.r_MaxDischargePowerAllowed := WORD_TO_REAL(MBMUData[45])-20000;			//-20k .. +20k kW in 1kW/bit steps
		
		BMSGet.MBMU_Status.BatteryStatus.r_SystemPower	:= 	WORD_TO_REAL(MBMUData[46])-20000;						//-20k .. +20k kW in 1kW/bit steps
		BMSGet.MBMU_Status.BatteryStatus.r_ChargeSOE	:=	WORD_TO_REAL(MBMUData[47])/10;
		BMSGet.MBMU_Status.BatteryStatus.r_DischargeSOE	:=	WORD_TO_REAL(MBMUData[48])/10;
		
		BMSGet.MBMU_Status.BatteryStatus.r_RemainingChargeEnergy	:=	WORD_TO_REAL(MBMUData[49]);
		BMSGet.MBMU_Status.BatteryStatus.r_RemainingDischargeEnergy	:=	WORD_TO_REAL(MBMUData[50]);
		
		BMSGet.MBMU_Status.BatteryStatus.r_MaxSystemVoltageAllowed := WORD_TO_REAL(MBMUData[51])/10; 			//0-1500V with 0.1V/bit
		BMSGet.MBMU_Status.BatteryStatus.r_MinSystemVoltageAllowed := WORD_TO_REAL(MBMUData[52])/10; 			//0-1500V with 0.1V/bit
		
		BMSGet.BattInfo := BMSGet.MBMU_Status.BatteryStatus;
		
		GetMBMUData := TRUE;
		COMretryCounter := 0;
	ELSE
		COMretryCounter := COMretryCounter +1;
		IF COMRetryCounter > 5 THEN
			b_MBComErrorActive := TRUE;
		END_IF
	END_IF
END_IF
END_METHOD

METHOD GetMBMUStaticSystemData : BOOL
VAR_INST
	MBReadBMS			: 	FB_MBReadRegs;
	DataBuffer 			: 	ARRAY[0..31] OF WORD;
	
	bCommBusy			:	BOOL;
	bComError			:	BOOL;
	errID				:	UDINT;
	cbRead				:	UDINT;
	
	TransmissionDone 	: 	f_trig;
	COMretryCounter		:	USINT := 0;
	ComTimer			:	Ton := (PT := TIME#200ms);
END_VAR

//Read ETH+MBMU SW/HW version at init.
GetMBMUStaticSystemData := FALSE;

ComTimer(in := NOT(ComTimer.Q));

MBReadBMS(
sIPAddr := Config.IP_BMS,
nTCPPort := Config.MBPort_BMS,
nUnitID := 255,//16#FF;
nMBAddr := 256,
nQuantity := 32,
cbLength := SIZEOF(DataBuffer),
pDestAddr := ADR(DataBuffer),
bExecute := ComTimer.Q,
tTimeout := T#100MS,
bBusy => bCommBusy,
bError => bComError,
nErrId => errID,
cbRead => cbRead
);

TransmissionDone(CLK := bCommBusy);

IF TransmissionDone.Q THEN
	IF NOT bComError THEN
		memcpy(destAddr := ADR(BMSGet.MBMU_Status.s_MBMU_SWVer), SrcAddr := ADR(DataBuffer[0]), n := 16);
		memcpy(destAddr  := ADR(BMSGet.MBMU_Status.s_MBMU_HWVer), SrcAddr := ADR(DataBuffer[8]), n := 16);
		memcpy(destAddr  := ADR(BMSGet.MBMU_Status.s_ETH_SWVer), SrcAddr := ADR(DataBuffer[16]), n := 16);
		memcpy(destAddr  := ADR(BMSGet.MBMU_Status.r_ETH_HWVer), SrcAddr :=ADR( DataBuffer[24]), n := 16);
		GetMBMUStaticSystemData := TRUE;
		COMretryCounter := 0;
	ELSE
		COMretryCounter := COMretryCounter +1;
		IF COMRetryCounter > 5 THEN
			b_MBComErrorActive := TRUE;
		END_IF
	END_IF
END_IF
END_METHOD

METHOD GetSBMUData : BOOL
VAR_INST
	MBReadSBMU		: 	FB_MBReadRegs;
	DataBuffer		:	ARRAY[0..87] OF WORD;
	bCommBusy		:	BOOL;
	bComError		:	BOOL;
	errID			:	UDINT;
	cbRead			:	UDINT;
	CommDone		: 	f_trig;
	
	SBMUCounter			: 	USINT	:=	0;
	COMretryCounter	:	USINT	:=	0;
	ComTimer			:	Ton := (PT := TIME#0S200MS);
END_VAR
GetSBMUData := FALSE;

ComTimer(in := NOT(ComTimer.Q));

MBReadSBMU(
	sIPAddr := Config.IP_BMS,
	nTCPPort := Config.MBPort_BMS,
	nUnitID := 255,//16#FF;
	nMBAddr := 1024*(SBMUcounter+1),
	nQuantity := 87,
	cbLength := SIZEOF(DataBuffer),
	pDestAddr := ADR(DataBuffer),
	bExecute := ComTimer.Q,
	tTimeout := TIME#100MS,
	bBusy => bCommBusy,
	bError => bComError,
	nErrId => errID,
	cbRead => cbRead
);
	
CommDone(CLK := bCommBusy);
	
IF CommDone.Q THEN
	IF NOT bComError THEN
		BMSGet.SBMU[SBMUcounter].w_SystemWarning := DataBuffer[0];
		BMSGet.SBMU[SBMUcounter].SystemAlarm[0] := DataBuffer[1];
		BMSGet.SBMU[SBMUcounter].SystemAlarm[1] := DataBuffer[2];
		BMSGet.SBMU[SBMUcounter].SystemAlarm[2] := DataBuffer[3];
		
		BMSGet.SBMU[SBMUcounter].b_PrechargeRelayClosed 	:= WORD_TO_BOOL(DataBuffer[16]);
		BMSGet.SBMU[SBMUcounter].b_MainPosRelayClosed	 	:= WORD_TO_BOOL(DataBuffer[17]);
		BMSGet.SBMU[SBMUcounter].b_MainNegRelayClosed		:= WORD_TO_BOOL(DataBuffer[18]);
		BMSGet.SBMU[SBMUcounter].b_ControlBoxFanOn 			:= WORD_TO_BOOL(DataBuffer[19]);
		BMSGet.SBMU[SBMUcounter].b_BalanceStatus 			:= WORD_TO_BOOL(DataBuffer[20]);
		
		BMSGet.SBMU[SBMUcounter].BatteryStatus.r_SystemVoltage := WORD_TO_REAL(DataBuffer[32])/10;	//0-1500V with 0.1V/bit
		BMSGet.SBMU[SBMUcounter].BatteryStatus.r_SystemCurrent := (WORD_TO_REAL(DataBuffer[34])/10)-2000; 	//-2k .. +2k A in 0.1A/bit steps
		
		BMSGet.SBMU[SBMUcounter].BatteryStatus.r_SOC := WORD_TO_REAL(DataBuffer[35])/10; 			//0-100% with 0.1%/bit;
		BMSGet.SBMU[SBMUcounter].BatteryStatus.r_SOH := WORD_TO_REAL(DataBuffer[36])/10;				//0-100% with 0.1%/bit;
		
		BMSGet.SBMU[SBMUcounter].BatteryStatus.CellVoltage[eSubValues.Maximum] := WORD_TO_REAL(DataBuffer[37])/1000;	//0-5v with 0.001v/bit;
		BMSGet.SBMU[SBMUcounter].BatteryStatus.CellVoltage[eSubValues.Average] := WORD_TO_REAL(DataBuffer[39])/1000;	//0-5v with 0.001v/bit;
		
		BMSGet.SBMU[SBMUcounter].BatteryStatus.CellTemperature[eSubValues.Maximum] := WORD_TO_REAL(DataBuffer[40])-50;	//-50..200gr with 1gr/bit;
		BMSGet.SBMU[SBMUcounter].BatteryStatus.CellTemperature[eSubValues.Minimum] := WORD_TO_REAL(DataBuffer[41])-50;	//-50..200gr with 1gr/bit;
		BMSGet.SBMU[SBMUcounter].BatteryStatus.CellTemperature[eSubValues.Average] := WORD_TO_REAL(DataBuffer[42])-50;	//-50..200gr with 1gr/bit;
		
		BMSGet.SBMU[SBMUcounter].BatteryStatus.r_MaxChargeCurrentAllowed := 		(WORD_TO_REAL(DataBuffer[43])/10)-2000;	//-2k .. +2k A in 0.1A/bit steps
		BMSGet.SBMU[SBMUcounter].BatteryStatus.r_MaxDischargeCurrentAllowed := 		(WORD_TO_REAL(DataBuffer[44])/10)-2000;	//-2k .. +2k A in 0.1A/bit steps
		
		BMSGet.SBMU[SBMUcounter].BatteryStatus.w_MaxVoltageCellLocation := DataBuffer[48];
		BMSGet.SBMU[SBMUcounter].BatteryStatus.w_MinVoltageCellLocation := DataBuffer[49];
		
		BMSGet.SBMU[SBMUcounter].BatteryStatus.w_MaxTempCellLocation := DataBuffer[50];
		BMSGet.SBMU[SBMUcounter].BatteryStatus.w_MinTempCellLocation := DataBuffer[51];
		
		BMSGet.SBMU[SBMUcounter].BatteryStatus.r_SumOfCellVoltages := WORD_TO_REAL(DataBuffer[55])/10;	//0-1500V with 0.1V/bit
		
		MEMCPY(ADR(BMSGet.SBMU[SBMUcounter].BatteryStatus.r_HistAccChargeEnergy), ADR(DataBuffer[85]), 2);  // low word
		MEMCPY(ADR(BMSGet.SBMU[SBMUcounter].BatteryStatus.r_HistAccChargeEnergy)+2, ADR(DataBuffer[84]), 2);  // high word
		BMSGet.SBMU[SBMUcounter].BatteryStatus.r_HistAccChargeEnergy := BMSGet.SBMU[SBMUcounter].BatteryStatus.r_HistAccChargeEnergy/10; //0-449GHW with 0.1kWh/bit
		
		MEMCPY(ADR(BMSGet.SBMU[SBMUcounter].BatteryStatus.r_HistAccDischargeEnergy), ADR(DataBuffer[87]), 2);  // low word
		MEMCPY(ADR(BMSGet.SBMU[SBMUcounter].BatteryStatus.r_HistAccDischargeEnergy)+2, ADR(DataBuffer[86]), 2);  // high word
		BMSGet.SBMU[SBMUcounter].BatteryStatus.r_HistAccDischargeEnergy := BMSGet.SBMU[SBMUcounter].BatteryStatus.r_HistAccDischargeEnergy/10; //0-449GHW with 0.1kWh/bit
	
		SBMUCounter := SBMUCounter +1;
		COMretryCounter := 0;
		
		IF SBMUCounter >= 4 THEN//BMSGet.MBMU_Status.by_NumberOfSubSystems THEN
			
			GetSBMUData := TRUE;
			SBMUCounter := 0;
		END_IF
		
		
		IF 		(BMSGet.SBMU[0].b_MainPosRelayClosed AND BMSGet.SBMU[0].b_MainNegRelayClosed) AND
				(BMSGet.SBMU[1].b_MainPosRelayClosed AND BMSGet.SBMU[1].b_MainNegRelayClosed) AND
				(BMSGet.SBMU[2].b_MainPosRelayClosed AND BMSGet.SBMU[2].b_MainNegRelayClosed) AND
				(BMSGet.SBMU[3].b_MainPosRelayClosed AND BMSGet.SBMU[3].b_MainNegRelayClosed) THEN
			PowerStatus := eHVDC_PowerStatus.On;
		ELSIF 	BMSGet.SBMU[SBMUcounter].b_PrechargeRelayClosed OR 
				BMSGet.SBMU[SBMUcounter].b_PrechargeRelayClosed OR 
				BMSGet.SBMU[SBMUcounter].b_PrechargeRelayClosed OR 
				BMSGet.SBMU[SBMUcounter].b_PrechargeRelayClosed THEN
			PowerStatus := eHVDC_PowerStatus.Precharging;
		ELSE
			PowerStatus := eHVDC_PowerStatus.Off;
		END_IF	
		
		BMSGet.SBMU[SBMUcounter].b_PrechargeRelayClosed 	:= WORD_TO_BOOL(DataBuffer[16]);
		BMSGet.SBMU[SBMUcounter].b_MainPosRelayClosed	 	:= WORD_TO_BOOL(DataBuffer[17]);
		BMSGet.SBMU[SBMUcounter].b_MainNegRelayClosed		:= WORD_TO_BOOL(DataBuffer[18]);
		BMSGet.SBMU[SBMUcounter].b_ControlBoxFanOn 			:= WORD_TO_BOOL(DataBuffer[19]);
		BMSGet.SBMU[SBMUcounter].b_BalanceStatus 			:= WORD_TO_BOOL(DataBuffer[20]);
	ELSE
		COMretryCounter := COMretryCounter +1;
		IF COMRetryCounter > 5 THEN
			b_MBComErrorActive := TRUE;
		END_IF
	END_IF
END_IF
END_METHOD

METHOD GetSBMUStaticSystemData : BOOL

VAR_INPUT
	SBMU_ID				:	uint;	
END_VAR

VAR_INST
	MBReadBMS			: 	FB_MBReadRegs;
	DataBuffer 			: 	ARRAY[0..31] OF WORD;
	
	bCommBusy			:	BOOL;
	bComError			:	BOOL;
	errID				:	UDINT;
	cbRead				:	UDINT;
	
	TransmissionDone 	: 	f_trig;
	ComretryCounter		:	USINT := 0;
	
	ComTimer			:	Ton := (PT := TIME#0S200MS);
END_VAR


VAR
	SBMU: INT;
END_VAR
//Read ETH+MBMU SW/HW version at init.
GetSBMUStaticSystemData := FALSE;

IF (SBMU_ID<1) OR (SBMU>4)then //BMSGET.MBMU_Status.by_NumberOfSubSystems) THEN
	GetSBMUStaticSystemData := TRUE;
	RETURN;
END_IF

ComTimer(in := NOT(ComTimer.Q));

MBReadBMS(
sIPAddr := Config.IP_BMS,
nTCPPort := Config.MBPort_BMS,
nUnitID := 255,//16#FF;
nMBAddr := 960 + (SBMU_ID*1024),
nQuantity := 32,
cbLength := SIZEOF(DataBuffer),
pDestAddr := ADR(DataBuffer),
bExecute := ComTimer.Q,
tTimeout := T#100MS,
bBusy => bCommBusy,
bError => bComError,
nErrId => errID,
cbRead => cbRead
);

TransmissionDone(CLK := bCommBusy);

IF TransmissionDone.Q THEN
	IF NOT bComError THEN
	//werkt niet. Bij de MBMU gek genoeg wel
	//	memcpy(destAddr := ADR(BMSGet.SBMU[SBMU_ID].s_SBMU_SWVer), SrcAddr := ADR(DataBuffer[0]), n := 16);
	//	memcpy(destAddr  := ADR(BMSGet.SBMU[SBMU_ID].s_SBMU_HWVer), SrcAddr := ADR(DataBuffer[8]), n := 16);
	//	memcpy(destAddr  := ADR(BMSGet.SBMU[SBMU_ID].s_CSC_SWVer), SrcAddr := ADR(DataBuffer[16]), n := 16);
	//	memcpy(destAddr  := ADR(BMSGet.SBMU[SBMU_ID].s_CSC_HWVer), SrcAddr := ADR(DataBuffer[24]), n := 16);
		GetSBMUStaticSystemData := TRUE;
		ComretryCounter := 0;
	ELSE
		COMretryCounter := COMretryCounter +1;
		IF COMRetryCounter > 5 THEN
			b_MBComErrorActive := TRUE;
		END_IF
	END_IF
END_IF
END_METHOD

METHOD GetSystemStatus : BOOL
VAR_INST
	MBReadBMS			: 	FB_MBReadRegs;
	DataBuffer 			: 	ARRAY[0..3] OF WORD;
	
	bCommBusy			:	BOOL;
	bComError			:	BOOL;
	errID				:	UDINT;
	cbRead				:	UDINT;
	
	TransmissionDone 	: 	f_trig;
	
	ComTimer			:	Ton := (PT := TIME#0S200MS);
	
	ComretryCounter	:	USINT := 0;
END_VAR

//Read general BMS status
GetSystemStatus := FALSE;

ComTimer(in := NOT(ComTimer.Q));

MBReadBMS(
sIPAddr := Config.IP_BMS,
nTCPPort := Config.MBPort_BMS,
nUnitID := 255,//16#FF;
nMBAddr := 769,
nQuantity := 4,
cbLength := SIZEOF(DataBuffer),
pDestAddr := ADR(DataBuffer),
bExecute := ComTimer.Q,
bBusy => bCommBusy,
bError => bComError,
nErrId => errID,
cbRead => cbRead,
tTimeout	:= T#100MS
);

TransmissionDone(CLK := bCommBusy);

IF TransmissionDone.Q THEN
	IF NOT bComError THEN
		CASE DataBuffer[0] OF
			0: BMSGet.MBMU_Status.BatteryStatus.ui_BMS_PowerOnStatus := ePowerOnStatus.Off;
			1: BMSGet.MBMU_Status.BatteryStatus.ui_BMS_PowerOnStatus := ePowerOnStatus.On;
			2: BMSGet.MBMU_Status.BatteryStatus.ui_BMS_PowerOnStatus := ePowerOnStatus.PowerOn_Fault;
			3: BMSGet.MBMU_Status.BatteryStatus.ui_BMS_PowerOnStatus := ePowerOnStatus.PowerOff_Fault;
		END_CASE
		
		BMSGet.BattInfo.ui_BMS_PowerOnStatus := BMSGet.MBMU_Status.BatteryStatus.ui_BMS_PowerOnStatus;
		
		CASE DataBuffer[1] OF
			0: BMSGet.MBMU_Status.BatteryStatus.ui_BMS_Status := eBMS_Status.Init;
			1: BMSGet.MBMU_Status.BatteryStatus.ui_BMS_Status := eBMS_Status.Normal;
			2: BMSGet.MBMU_Status.BatteryStatus.ui_BMS_Status := eBMS_Status.FullCharge;
			3: BMSGet.MBMU_Status.BatteryStatus.ui_BMS_Status := eBMS_Status.FullDischarge;
			4: BMSGet.MBMU_Status.BatteryStatus.ui_BMS_Status := eBMS_Status.Warning;
			5: BMSGet.MBMU_Status.BatteryStatus.ui_BMS_Status := eBMS_Status.Fault;
		END_CASE
		
		BMSGet.BattInfo.ui_BMS_Status := BMSGet.MBMU_Status.BatteryStatus.ui_BMS_Status;
		
		BMSGet.MBMU_Status.by_NumberOfSubSystems := WORD_TO_BYTE(DataBuffer[3]);
		GetSystemStatus := TRUE;
		ComretryCounter := 0;
	ELSE
		COMretryCounter := COMretryCounter +1;
		IF COMRetryCounter > 5 THEN
			b_MBComErrorActive := TRUE;
		END_IF
	END_IF
END_IF
END_METHOD

METHOD OpenInsulationSwitch : BOOL
VAR_INPUT
	OpenSwitch : BOOL;
END_VAR

VAR_INST
	WriteReg	:	FB_MBWriteSingleReg;
	Value 		:	WORD 	:= 0;
	StartWrite	:	BOOL	:= FALSE;
	
	bCommBusy	:	BOOL;
	bComError	:	BOOL;
	errID		:	UDINT;

	TransmissionDone 	: 	f_trig;
	ComRetryCounter	:	USINT;
	
	ComTimer			:	Ton := (PT := TIME#0S200MS);
END_VAR

ComTimer(in := NOT(ComTimer.Q));

OpenInsulationswitch := FALSE;

IF OpenSwitch THEN
	Value := 1;
ELSE
	Value := 0;
END_IF

WriteReg(
sIPAddr := Config.IP_BMS,
nTCPPort := Config.MBPort_BMS,
nUnitID := 255,//16#FF;
nMBAddr := 907,
nValue := Value,
tTimeout := T#0S100MS,
bExecute := ComTimer.q,
bBusy => bCommBusy,
bError => bComError,
nErrId => errID,
);

TransmissionDone(CLK := bCommBusy);

IF TransmissionDone.Q THEN
	IF NOT bComError THEN
		BMSGet.MBMU_Status.b_InsulationSwitchOpen := OpenSwitch;
		ComRetryCounter := 0;
		OpenInsulationSwitch := TRUE;
	ELSE
		COMretryCounter := COMretryCounter +1;
		IF COMRetryCounter > 5 THEN
			b_MBComErrorActive := TRUE;
		END_IF
	END_IF
END_IF
END_METHOD

METHOD Reset : BOOL
VAR_INPUT
	//BMSSET	:	st_BMS_Set;
	//ResetIn	:	BOOL;
END_VAR

VAR_INST
	ResetTrigger		:	Ton := (PT := TIME#1S0MS);
	ResetVar			:	BOOL;
END_VAR
Reset := FALSE;

IF FBState = ePOUState.Normal OR FBState = ePOUState.EMSTOP THEN
	IF ClearBMSFaults() THEN
		FBState := ePOUState.Normal;
	END_IF
END_IF
END_METHOD

METHOD SetBMSDateTime : BOOL
VAR
	SystemTimeData	:	Timestruct;
	RTCData	:	ARRAY[0..6] OF WORD;	
	
END_VAR
VAR_INST
	ComTimer			:	Ton := (PT := TIME#0S200MS);
	WriteRegs		:	FB_MBWriteRegs;
	SystemTime		:	FB_LocalSystemTime;
	TransmissionDone 	: 	f_trig;
	SystemTimeDataValid	:	BOOL;
	bCommBusy		:	BOOL;
	bComError		:	BOOL;
	errID			:	UDINT;
	COMRetryCounter	:	USINT := 0;
END_VAR
ComTimer(in := NOT(ComTimer.Q));

//write PLC system time to BMS RTC
SetBMSDateTime := FALSE;


//retrieve system time struct
SystemTime(
	sNetID := '',
	bEnable := TRUE,
	dwCycle := 1,
	dwOpt	:= 1,
	tTimeout := TIME#500MS,
	bValid => SystemtimeDataValid,
	systemTime => SystemTimeData
);

//parse system time to BMS data array
IF SystemTimeDataValid THEN
	RTCData[0] := 2024;//SystemTimeData.wYear;
	RTCData[1] := 03;//SystemTimeData.wMonth;
	RTCData[2] := 26;//SystemTimeData.wDay;
	RTCData[3] := 13;//SystemTimeData.wHour;
	RTCData[4] := 52;//SystemTimeData.wMinute;
	RTCData[5] := 00;//SystemTimeData.wSecond;
	RTCData[6] := 1;//can this value remain at 1? or reset to 0 after write?
	
	//write data to BMS
	WriteRegs(	
	sIPAddr := Config.IP_BMS,
	nTCPPort := Config.MBPort_BMS,
	nUnitID := 255,//16#FF;
	nMBAddr := 900,
	nQuantity := 7,
	pSrcAddr := ADR(RTCData),
	cbLength := SIZEOF(RTCData),
	bExecute := ComTimer.Q,
	tTimeout := TIME#100MS,
	bBusy => bCommBusy,
	bError => bComError,
	nErrId => errID,
	);
	
	TransmissionDone(CLK := bCommBusy);
	
	//return true if tranmission succeeds
	IF TransmissionDone.Q THEN
		IF NOT bComError THEN
			SetBMSDateTime := TRUE;
			ComRetryCounter := 0;
		ELSE
			COMretryCounter := COMretryCounter +1;
			IF COMRetryCounter > 5 THEN
				b_MBComErrorActive := TRUE;
			END_IF
		END_IF
	END_IF
END_IF
END_METHOD

METHOD SetPowerMode : BOOL
VAR_INST
	WriteReg	:	FB_MBWriteSingleReg;
	Value 		:	WORD 	:= 1;
	StartWrite	:	BOOL	:= FALSE;
	bCommBusy	:	BOOL;
	bComError	:	BOOL;
	errID		:	UDINT;
	TransmissionDone 	: 	f_trig;
	ComTrigger	:	Ton := (PT := TIME#200MS);
	ComRetryCounter	:	USINT	:= 0;
END_VAR	

VAR

END_VAR

Value := ePowerControl.Stay; //default command is: Do nothing
//it may also work if we just keep sending "poweron" if b_HVDC_Required is true. But this doesn't seem to be the way they intended.

IF Set.b_HVDC_Required AND (BMSGet.BattInfo.ui_BMS_PowerOnStatus = ePowerOnStatus.Off) THEN	//send poweron if system not already on
	Value := ePowerControl.PowerOn;
ELSIF (NOT Set.b_HVDC_Required) AND (BMSGet.BattInfo.ui_BMS_PowerOnStatus = ePowerOnStatus.On) THEN //send poweroff if system not already off
	Value := ePowerControl.PowerOff;
END_IF

//Write this register every second, regardless of change.
ComTrigger(in := NOT(ComTrigger.Q));

//IF BMSGet.BattInfo.ui_BMS_Status < 5 THEN
WriteReg(
	sIPAddr := Config.IP_BMS,
	nTCPPort := Config.MBPort_BMS,
	nUnitID := 255,//16#FF;
	nMBAddr := 897,
	nValue := Value,
	tTimeout := T#0S100MS,
	bExecute := ComTrigger.Q,
	bBusy => bCommBusy,
	bError => bComError,
	nErrId => errID,
);
//ELSE
//	SetPowerMode := TRUE;
//END_IF

	
TransmissionDone(CLK := bCommBusy);
	
//return true if tranmission succeeds
IF TransmissionDone.Q THEN
	IF NOT bComError THEN
		SetPowerMode := TRUE;
		ComRetryCounter := 0;
	ELSE
		COMretryCounter := COMretryCounter +1;
		IF COMRetryCounter > 5 THEN
			b_MBComErrorActive := TRUE;
		END_IF
	END_IF
END_IF
END_METHOD

ACTION SFCTipReset:
SFCTip := FALSE;
END_ACTION

END_FUNCTION_BLOCK

(* stored: Version 1.1.0.1, ProductVersion 3.1.4024.12
   POU FB_BMS: Id {5a961730-f4bc-46e9-979d-c80cbcef2de5}, SpecialFunc None
   Folder Internal methods: Id {0651177a-376e-46f3-b8bb-dfd934f25570}
   Folder SFC: Id {22c86a39-5de5-4c8d-b9fe-00d65834d86f}
   Action aBMSPoweroff: Id {05a3f9df-6ae0-4bcb-ae8e-855375a58730}
   Action aBMSPowerOn: Id {3743f205-15b2-408e-8a62-6f783ffd0641}
   Action aClearFaults: Id {9c7e4fd3-e0fe-411d-b59c-f3f1361caeaf}
   Action aDisableInsulationMonitor: Id {ce418a82-36be-4340-9296-5bcd738823d9}
   Action aGetMBMUData: Id {4d3b6c31-cb9f-4968-b7ae-31e81eb63d9b}
   Action aGetSBMUData: Id {938e7840-1309-4050-aeed-115b8e1c45d4}
   Action aGetStaticData: Id {72e4a65b-ace1-4c9c-8f3b-95f864b6c151}
   Action aGetStatus: Id {aa8f426c-f58f-4996-878b-62e4a336c3d9}
   Action aInit: Id {185800e8-9ce9-49b6-8e1a-efe2e0c8c813}
   Action aSetDateTime: Id {5afb45d8-c9b4-48b4-8b6d-cd0fce31ca0f}
   Action aSetPowerMode: Id {c0cb5012-948e-4d4c-a5f7-7892e11c8df2}
   Action aWatchdog: Id {3d838ac5-e3d0-4374-af5d-b5c243be25cc}
   Method BMS_Diagnostics: Id {e54d08a6-45aa-4c23-a639-a7e2c50802a6}
   Method BMSHeartBeat: Id {00b15e11-892f-4f1a-9ab4-2fe4dc92a7ec}
   Action BMSSFC: Id {5f839ee7-6432-4da8-b44e-b2774bd29b0b}
   Method ClearBMSFaults: Id {dd3f73ff-65b4-4d34-a987-bf3c7898eed7}
   Method EMSTOP: Id {2604fb3b-f967-4753-838f-b4c74bb783ff}
   Method GetCellData: Id {c8c431ea-294f-491e-8003-5ad2a08d370c}
   Method GetDiagnostics: Id {6224be93-201c-4c60-b282-164718f1984c}
   Method GetMBMUData: Id {677deb29-d719-4389-9493-1039376b0db6}
   Method GetMBMUStaticSystemData: Id {bac0e602-85b6-4537-9145-8883fc8dca2f}
   Method GetSBMUData: Id {7c92f7c9-c74b-4dce-aa1b-db05b97f85d3}
   Method GetSBMUStaticSystemData: Id {fd82471a-3a1b-48e3-8c3c-308812129576}
   Method GetSystemStatus: Id {a90d1736-4794-4e09-9309-5d9b0bd48118}
   Method OpenInsulationSwitch: Id {222ceca3-fad3-4e38-899f-8fd91baeacf6}
   Method Reset: Id {276c673a-6724-4959-86e2-577bb9e79adb}
   Method SetBMSDateTime: Id {10061d03-20f6-4f95-aa91-0bfb4aa16ea7}
   Method SetPowerMode: Id {b51b911d-6da4-4232-b339-d545e512eeeb}
   Action SFCTipReset: Id {bd39e870-0e61-4d10-baf7-1dc4d7417da6} *)
